FUNCTION FC_GetCurrentCycleCount : UDINT

FC_GetCurrentCycleCount := IING.cycleCounter;

END_FUNCTION

(* stored: Version 1.1.0.1, ProductVersion 3.1.4026.18
   POU FC_GetCurrentCycleCount: Id {5a00b2cc-ec1a-4990-a2eb-0f3fd85f519f}, SpecialFunc None *)
